FUNCTION_BLOCK Bedroom
VAR_INPUT
END_VAR
VAR_OUTPUT
END_VAR
VAR
END_VAR

END_FUNCTION_BLOCK

(* stored: Version 1.1.0.1, ProductVersion 3.1.4024.13
   POU Bedroom: Id {29421c85-e58d-4919-8d8f-6e5374a848f0}, SpecialFunc None *)
